FUNCTION_BLOCK FB_FMS205_SFC
VAR_INPUT
	IC: BOOL;
	Execute: BOOL;
	Ack: BOOL;
END_VAR
VAR_OUTPUT
	Ready: BOOL;
	Failure: BOOL;
	Done: BOOL;
END_VAR

VAR_IN_OUT
	mdAlimentador			: FB_Alimentador;
	mdPickAndPlaceCarga 	: FB_PickAndPlace;
	mdMedidorTapa			: FB_MedidorTapa;
	mdCaptadorInductivo 	: FB_CaptadorInductivo;
	mdDetectorFotoelectrico : FB_DetectorFotoelectrico;
	mdEvacuador			 	: FB_Evacuador;
	mdPickAndPlaceDescarga 	: FB_PickAndPlace;
	mdPlatoDivisor			: FB_PlatoDivisor;
	mdCinta					: FB_Cinta;
END_VAR
// TODO PENDIENTE TERMINAR EL RESTO DE MÓDULOS
VAR
END_VAR

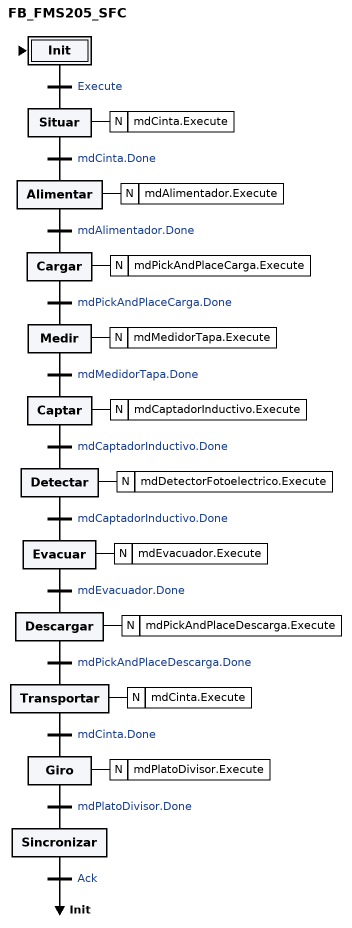
INITIAL_STEP Init:
END_STEP
TRANSITION FROM Init TO Situar
    := Execute;
END_TRANSITION
STEP Situar:
    mdCinta.Execute(N);
END_STEP
TRANSITION FROM Situar TO Alimentar
    := mdCinta.Done;
END_TRANSITION
STEP Alimentar:
    mdAlimentador.Execute(N);
END_STEP
TRANSITION FROM Alimentar TO Cargar
    := mdAlimentador.Done;
END_TRANSITION
STEP Cargar:
    mdPickAndPlaceCarga.Execute(N);
END_STEP
TRANSITION FROM Cargar TO Medir
    := mdPickAndPlaceCarga.Done;
END_TRANSITION
STEP Medir:
    mdMedidorTapa.Execute(N);
END_STEP
TRANSITION FROM Medir TO Captar
    := mdMedidorTapa.Done;
END_TRANSITION
STEP Captar:
    mdCaptadorInductivo.Execute(N);
END_STEP
TRANSITION FROM Captar TO Detectar
    := mdCaptadorInductivo.Done;
END_TRANSITION
STEP Detectar:
    mdDetectorFotoelectrico.Execute(N);
END_STEP
TRANSITION FROM Detectar TO Evacuar
    := mdCaptadorInductivo.Done;
END_TRANSITION
STEP Evacuar:
    mdEvacuador.Execute(N);
END_STEP
TRANSITION FROM Evacuar TO Descargar
    := mdEvacuador.Done;
END_TRANSITION
STEP Descargar:
    mdPickAndPlaceDescarga.Execute(N);
END_STEP
TRANSITION FROM Descargar TO Transportar
    := mdPickAndPlaceDescarga.Done;
END_TRANSITION
STEP Transportar:
    mdCinta.Execute(N);
END_STEP
TRANSITION FROM Transportar TO Giro
    := mdCinta.Done;
END_TRANSITION
STEP Giro:
    mdPlatoDivisor.Execute(N);
END_STEP
TRANSITION FROM Giro TO Sincronizar
    := mdPlatoDivisor.Done;
END_TRANSITION
STEP Sincronizar:
END_STEP
TRANSITION FROM Sincronizar TO Init
    := Ack;
END_TRANSITION

END_FUNCTION_BLOCK

(* stored: Version 1.1.0.1, ProductVersion 3.1.4024.6
   POU FB_FMS205_SFC: Id {a81c472c-1220-4b76-860b-f7f6b111694f}, SpecialFunc None *)
